FUNCTION F_GetDefaultMainBlade : ST_SawBladeData
VAR_INPUT
END_VAR
VAR
END_VAR

F_GetDefaultMainBlade.rBladeDiameter := 350.0;
F_GetDefaultMainBlade.rBladeRadius := F_GetDefaultMainBlade.rBladeDiameter / 2;
F_GetDefaultMainBlade.rBladeThickness := 3.2;
F_GetDefaultMainBlade.sBladeType := 'TCT Panel Saw Blade PI-521VS Premium';

END_FUNCTION

(* stored: Version 1.1.0.1
   POU F_GetDefaultMainBlade: Id {ce87e513-ac8d-49c8-a43a-2c95bf2bc0e3}, SpecialFunc None *)
